FUNCTION UpdateEventTimestampWithSystemTime
VAR_INPUT
	stEvent : REFERENCE TO ST_Event;
	
END_VAR
VAR
	//fGetSystemTime : F_GetSystemTime; //实例化
	(*stFileTime : FILETIME64_TO_DT; //实例化，需要再reference中加入相关引用*)
	timeAsFileTime : T_FILETIME64;
	(*timeAsDT : DT;*)
END_VAR

timeAsFileTime := F_GetSystemTime();
stEvent.dtTimeStamp := FILETIME64_TO_DT(timeAsFileTime);

END_FUNCTION

(* stored: Version 1.1.0.1, ProductVersion 3.1.4024.12
   POU UpdateEventTimestampWithSystemTime: Id {5235ad37-4cf3-4d23-b79c-79031989d273}, SpecialFunc None *)
